INTERFACE I_TankController

METHOD ApplyCooling 
VAR_INPUT
END_VAR
END_METHOD

METHOD CheckSafety 
VAR_INPUT
END_VAR
END_METHOD

END_INTERFACE

(* stored: Version 1.1.0.1, ProductVersion 3.1.4024.16
   Itf I_TankController: Id {2dbfb90e-ccdf-4cc7-97b3-cf650202c10d}
   Method ApplyCooling: Id {58b5313a-dd06-4534-a521-4b12f93fd578}
   Method CheckSafety: Id {0190ea31-5b65-4a18-b434-2b5926760da6} *)
